# EPICS substitutions: pgpCamlinkApp/camera_config/Basler_acA2040-180kmNIR.substitutions
# A simple MODEL substitutions file which preserves macro defaults
# but expands any inluded rbvMonitor.template or other templates.
file Basler_acA2040-180kmNIR.template
{
	{
		P				= "\$(P)",
		R				= "\$(R)",
		PORT			= "\$(PORT)",
		PWIDTH			= "\$(PWIDTH=TRIG:PULSE:WIDTH)",
		PW_SCALE		= "\$(PW_SCALE=1e6)",
		SerialDisable	= "\$(SerialDisable)"
	}
}
